{attribute 'qualified_only'}
{attribute 'strict'}
{attribute 'to_string'}
TYPE EN_AtlasPumpAction :
(
    IDLE := 0,
    STOP_LEFT,
	STOP_RIGHT,
    PAUSE_LEFT,
    PAUSE_RIGHT,
	UNPAUSE_LEFT,
	UNPAUSE_RIGHT,
    EMPTY_LEFT_FAST,
    EMPTY_RIGHT_FAST,
    FILL_LEFT_FAST,
    FILL_RIGHT_FAST,
	EMPTY_LEFT_PRIME,
    EMPTY_RIGHT_PRIME,
    FILL_LEFT_PRIME,
    FILL_RIGHT_PRIME
);
END_TYPE

(* stored: Version 1.1.0.1
   DUT EN_AtlasPumpAction: Id {47914238-1076-04f0-16cb-edaecf0e8d21} *)
